RoboDK station: SingleRobot.rdk

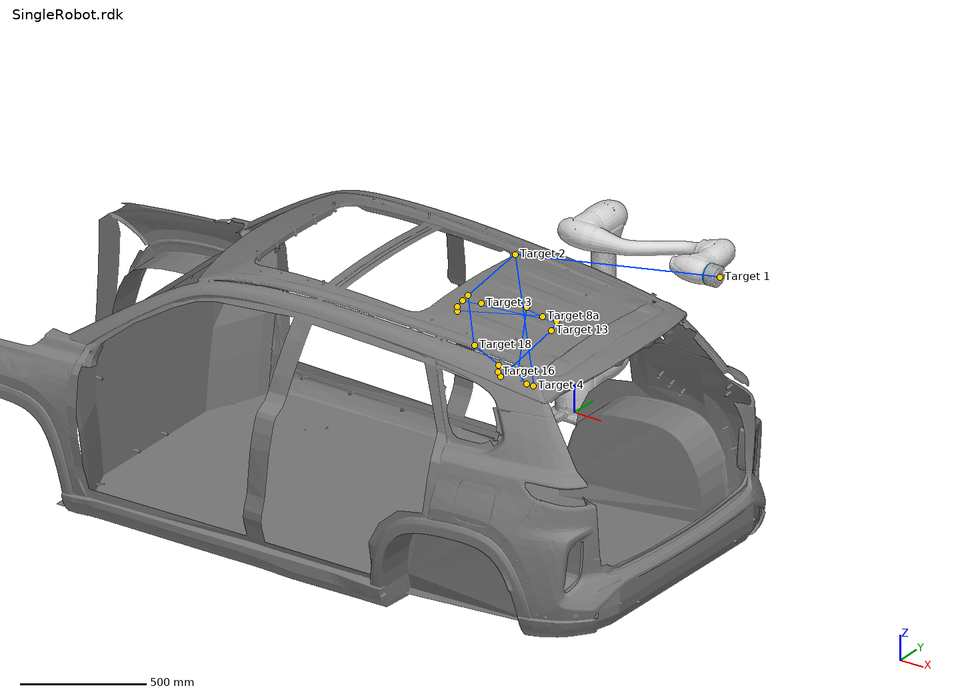
[picture v0: the station drawn from its stored meshes, robots at their saved joint values, targets as dots, program paths as lines]
Station SingleRobot (saved by RoboDK 6.0.4). Poses are relative to the parent item; angles as X-Y-Z fixed-axis rotations.
Station parameters (name, value as stored): CollisionFreePlanner, Doosan Robotics M1013 White, CollisionFreePlanner-Rob Doosan Robotics M1013 White
  - frame Doosan Robotics M1013 White Base at (401.74, 1165.46, 0) mm
    - robot Doosan Robotics M1013 White: 6 axes, payload 10 kg, reach 1300 mm, repeatability 0.05 mm, weight 33 kg
        modified DH rows (alpha deg, a mm, theta deg, d mm): 0, 0, 0, 152.5; -90, 0, -90, -34.506; 0, 620, -90, 0; -90, 0, 0, 559; 90, 0, 0, 0; -90, 0, 180, 121
        base shift (0, 0, 0) mm, rotated rx 0 ry 0 rz 180 deg
        joint limits [-360, -360, -160, -360, -360, -360] to [360, 360, 160, 360, 360, 360]; home [0, 0, 90, 0, 0, 0]; saved at [0, 0, 90, 0, 0, 0]
      - tool Tool 1, TCP at (0, 0, 0) mm
    - target Target 1 (Cartesian target) at (680, 34.51, 772.5) mm, rotated rx 0 ry 90 rz 0 deg; joints [0, 0, 90, 0, 0, 0] of Doosan Robotics M1013 White
    - target Target 2 (Cartesian target) at (103.09, -555.05, 945.96) mm, rotated rx -5.44 ry 9.33 rz -85.51 deg; joints [-84.1, -1.24, 85.62, -5.39, -74.98, 0] of Doosan Robotics M1013 White
    - target Target 3 (Cartesian target) at (131.23, -827.38, 847.54) mm, rotated rx -5.55 ry 13.92 rz -85.54 deg; joints [-84.1, 23.61, 65.36, -5.39, -74.98, 0] of Doosan Robotics M1013 White
    - target Target 4 (Cartesian target) at (421.79, -882.77, 588.52) mm, rotated rx -110.13 ry -18.39 rz -121.99 deg; joints [-69.98, 31.07, 64.63, -116.44, -33.36, 0] of Doosan Robotics M1013 White
    - target Target 5 (Cartesian target) at (403, -905.55, 599.74) mm, rotated rx -104.7 ry -22.91 rz -137.28 deg; joints [-69.98, 31.07, 64.63, -116.44, -18.36, 0] of Doosan Robotics M1013 White
    - target Target 6 (Cartesian target) at (376.89, -926.06, 650.25) mm, rotated rx -93.69 ry -26.33 rz -157.12 deg; joints [-69.98, 31.07, 61.63, -116.44, -1.36, 0] of Doosan Robotics M1013 White
    - target Target 7 (Cartesian target) at (376.98, -865.6, 913.9) mm, rotated rx -72.75 ry -14.4 rz -152.77 deg; joints [-69.98, 29.07, 41.63, -101.44, -11.36, 0] of Doosan Robotics M1013 White
    - target Target 8 (Cartesian target) at (329.34, -878.88, 923.13) mm, rotated rx -68.55 ry -6.33 rz -175.77 deg; joints [-69.98, 29.07, 41.63, -101.44, 12.64, 0] of Doosan Robotics M1013 White
    - target Target 8a (Cartesian target) at (419.53, -819.29, 867.31) mm, rotated rx -43.43 ry 4 rz -84.39 deg; joints [-69.97, 33.06, 45.85, -44.33, -69.18, 0] of Doosan Robotics M1013 White
    - target Target 9 (Cartesian target) at (119.19, -977.85, 870.85) mm, rotated rx 64.36 ry -3.7 rz -41.44 deg; joints [-79.97, 39.07, 31.63, 72.41, -49.3, 0] of Doosan Robotics M1013 White
    - target Target 10 (Cartesian target) at (85.59, -930.9, 861.24) mm, rotated rx 68.69 ry -15.06 rz -67.42 deg; joints [-79.96, 39.06, 31.63, 72.41, -77.29, 0] of Doosan Robotics M1013 White
    - target Target 11 (Cartesian target) at (86.65, -893.89, 874.12) mm, rotated rx 60.9 ry -20.09 rz -81.41 deg; joints [-79.95, 39.06, 31.62, 60.41, -91.58, 0] of Doosan Robotics M1013 White
    - target Target 11a (Cartesian target) at (105.56, -883.24, 899.91) mm, rotated rx 44.71 ry -19.84 rz -80.48 deg; joints [-79.94, 39.05, 31.62, -135.47, 90.72, 179.99] of Doosan Robotics M1013 White
    - target Target 12 (Cartesian target) at (414.34, -715.64, 802.41) mm, rotated rx -111.86 ry -9.86 rz -53.31 deg; joints [-69.98, 29.07, 45.11, -108.12, -107.3, 0] of Doosan Robotics M1013 White
    - target Target 13 (Cartesian target) at (418.24, -758, 779.2) mm, rotated rx -125.4 ry -15.08 rz -68.88 deg; joints [-69.98, 29.07, 45.1, -125.11, -91.3, 0] of Doosan Robotics M1013 White
    - target Target 15 (Cartesian target) at (266.81, -887.89, 587.08) mm, rotated rx -112.93 ry 9.04 rz 144.27 deg; joints [-69.97, 29.05, 67.2, -66.2, 52.6, 0] of Doosan Robotics M1013 White
    - target Target 16 (Cartesian target) at (243.9, -874.28, 596.45) mm, rotated rx -107.83 ry 1.41 rz 134.26 deg; joints [-69.98, 29.06, 67.2, -73.21, 64.61, 0] of Doosan Robotics M1013 White
    - target Target 17 (Cartesian target) at (214.61, -826.01, 599.28) mm, rotated rx -106.61 ry -6.71 rz 108.48 deg; joints [-69.97, 29.05, 67.2, -73.21, 91.61, 0] of Doosan Robotics M1013 White
    - target Target 18 (Cartesian target) at (95.8, -824.6, 651.69) mm, rotated rx -114.25 ry -9.23 rz 77.81 deg; joints [-78.97, 31.05, 57.2, -64.21, 115.61, 0] of Doosan Robotics M1013 White
  - object Hyryder chasis_extra studs at (0, -1.39, -0.47) mm, rotated rx 90 ry 0 rz 180 deg, size 3494.4 x 1172.8 x 1532.6 mm, geometry from Hyryder chasis_extra studs.obj
  - camera Camera 1
  - program Prog1 (23 instructions, listed below)
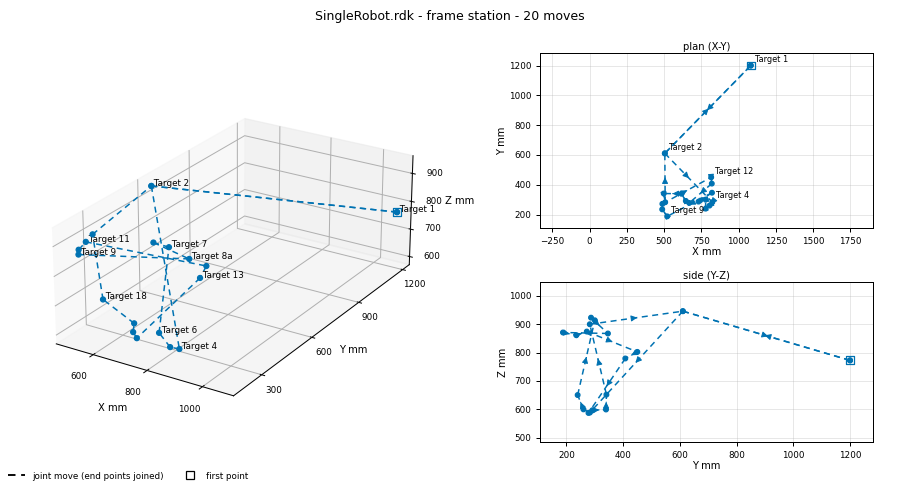
[picture p0: tool path of SingleRobot.rdk in frame station, 20 of 20 moves have a stored position in this frame; points joined in program order, loops and branches not executed]

--- program Prog1 (robot Doosan Robotics M1013 White) ---
  Set Ref.: Doosan Robotics M1013 White Base
  Set speed (0.5 mm/s)
  Set Tool: Tool 1
  MoveJ (Target 1)
  MoveJ (Target 2)
  MoveJ (Target 4)
  MoveJ (Target 5)
  MoveJ (Target 6)
  MoveJ (Target 7)
  MoveJ (Target 8)
  MoveJ (Target 8a)
  MoveJ (Target 9)
  MoveJ (Target 10)
  MoveJ (Target 11)
  MoveJ (Target 12)
  MoveJ (Target 13)
  MoveJ (Target 15)
  MoveJ (Target 16)
  MoveJ (Target 17)
  MoveJ (Target 18)
  MoveJ (Target 19) -> target Target 11a
  MoveJ (Target 2)
  MoveJ (Target 1)
